{attribute 'linkalways'} 
{attribute 'no_explicit_call' := 'This FB is a CLASS and must be accessed using methods or properties'}
{attribute 'enable_dynamic_creation'}
FUNCTION_BLOCK Node_F_VN_FillContainerExp_TcVnVector3_INT EXTENDS VisionNode
VAR
    ipContainer : _ITcVnContainer;
    aValue : _TcVnVector3_INT;
    nStartIdx : _ULINT(0);
    nCount : _ULINT(0);
    hrPrev : _HRESULT(S_OK);
    hresult : _HRESULT(S_OK);
END_VAR

METHOD PUBLIC  Clone : I_Node
VAR
    pNode : POINTER TO Node_F_VN_FillContainerExp_TcVnVector3_INT;
END_VAR
pNode := __NEW(Node_F_VN_FillContainerExp_TcVnVector3_INT);
Clone := pNode^;
END_METHOD

METHOD FB_init : BOOL
VAR_INPUT
    bInitRetains : BOOL; // if TRUE, the retain variables are initialized (warm start / cold start)
    bInCopyCode : BOOL;  // if TRUE, the instance afterwards gets moved into the copy code (online change)
END_VAR
AddInput('ipContainer', ipContainer);
AddInput('aValue', aValue);
AddInput('nStartIdx', nStartIdx);
AddInput('nCount', nCount);
AddInput('hrPrev', hrPrev);
AddOutput('ipContainer', ipContainer);
AddOutput('hresult',hresult);
END_METHOD

METHOD PROTECTED OnExecute : HRESULT
hresult.Value := F_VN_FillContainerExp_TcVnVector3_INT(
    ipContainer := ipContainer.Value,
    aValue := aValue.Value,
    nStartIdx := nStartIdx.Value,
    nCount := nCount.Value,
    hrPrev:= hrPrev.Value);
END_METHOD

METHOD PUBLIC PreExecutionCheck
VAR_INPUT
    Check : I_PreExecutionChecks;
END_VAR
Check.IsTrue(ipContainer.IsValid, 'ipContainer must be a valid container');
Check.IsTrue(ipContainer.HasType(TC_GLOBAL_CONST_LIST.ContainerType_Vector_TcVnVector3_INT), 'ipContainer contains incorrect type');
END_METHOD

END_FUNCTION_BLOCK

(* stored: Version 1.1.0.1, ProductVersion 3.1.4024.13
   POU Node_F_VN_FillContainerExp_TcVnVector3_INT: Id {83373cbe-54c8-4f49-84dc-eb8e17e173fc}, SpecialFunc None
   Folder Constructor: Id {9a216aea-3aa7-428d-b3f0-a53e260a5df3}
   Method Clone: Id {911bfd40-8ddf-40a6-99d9-500556dfd3d2}
   Method FB_init: Id {32e2a510-4d43-452f-8ebe-c178549ec4a4}
   Method OnExecute: Id {00adce3c-682f-4980-8415-d72274011fa9}
   Method PreExecutionCheck: Id {634fb4b8-53f5-493b-aabf-2cf8eed351be} *)
